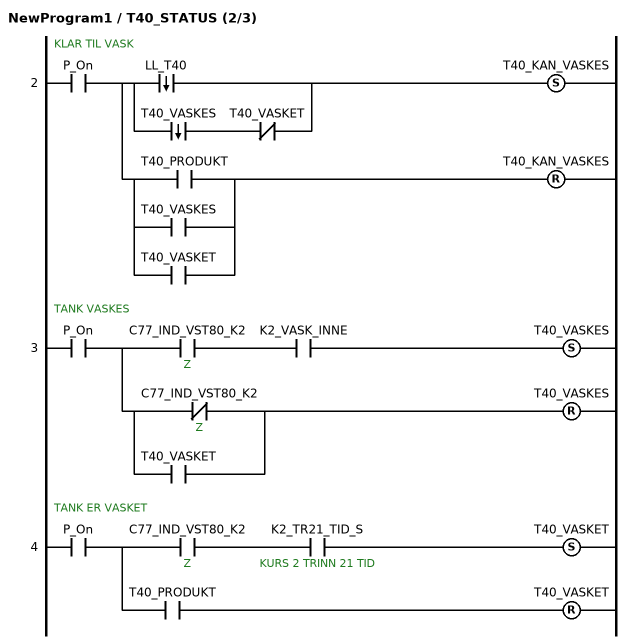
; [picture p1008: NewProgram1 / T40_STATUS, rungs 2-4]
; rung 2: KLAR TIL VASK
LD P_On
OUT TR0
%LD LL_T40
%LD T40_VASKES
ANDNOT T40_VASKET
ORLD
ANDLD
SET T40_KAN_VASKES
LD TR0
LD T40_PRODUKT
OR T40_VASKES
OR T40_VASKET
ANDLD
RSET T40_KAN_VASKES
; rung 3: TANK VASKES
LD P_On
OUT TR0
AND C77_IND_VST80_K2  ; Z
AND K2_VASK_INNE
SET T40_VASKES
LD TR0
LDNOT C77_IND_VST80_K2  ; Z
OR T40_VASKET
ANDLD
RSET T40_VASKES
; rung 4: TANK ER VASKET
LD P_On
OUT TR0
AND C77_IND_VST80_K2  ; Z
AND K2_TR21_TID_S  ; KURS 2 TRINN 21 TID
SET T40_VASKET
LD TR0
AND T40_PRODUKT
RSET T40_VASKET

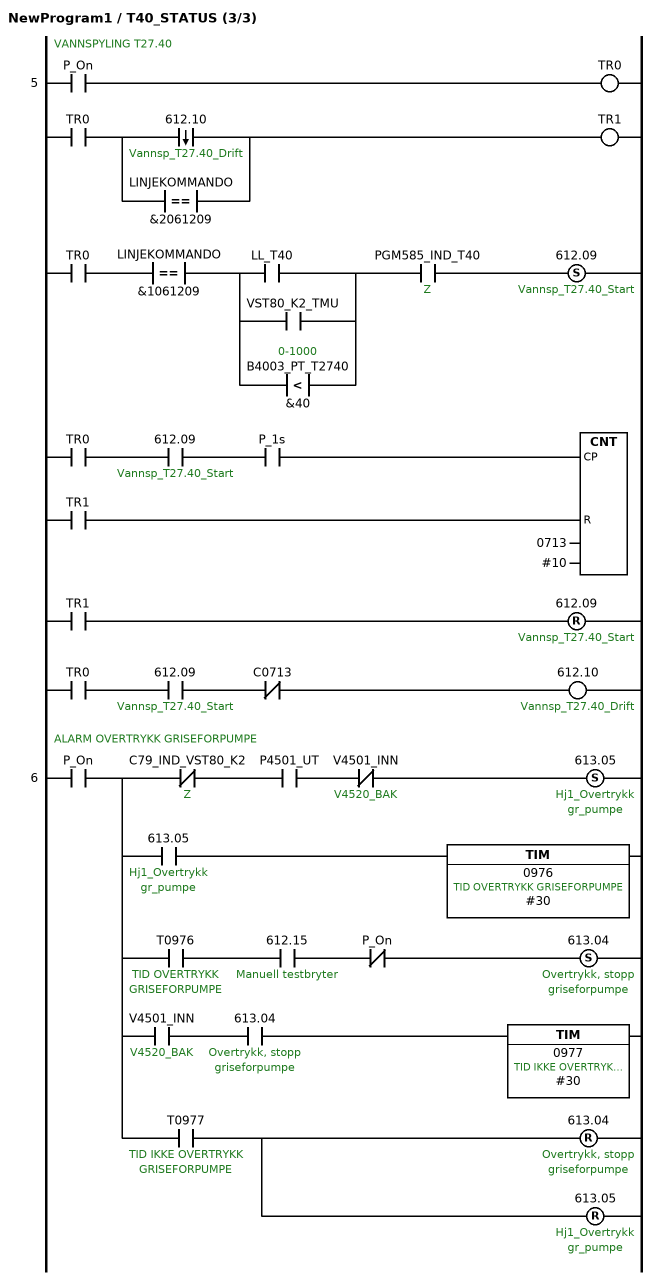
; rung 5: VANNSPYLING T27.40
LD P_On
OUT TR0
AND=L(301) LINJEKOMMANDO &1061209
LD LL_T40
OR VST80_K2_TMU
OR<(310) B4003_PT_T2740 &40  ; 0-1000
ANDLD
AND PGM585_IND_T40  ; Z
SET 612.09  ; Vannsp_T27.40_Start
LD TR0
AND 612.09  ; Vannsp_T27.40_Start
AND P_1s
LD TR0
%LD 612.10  ; Vannsp_T27.40_Drift
OR=L(301) LINJEKOMMANDO &2061209
ANDLD
OUT TR1
CNT 0713 #10
LD TR1
RSET 612.09  ; Vannsp_T27.40_Start
LD TR0
AND 612.09  ; Vannsp_T27.40_Start
ANDNOT C0713
OUT 612.10  ; Vannsp_T27.40_Drift
; rung 6: ALARM OVERTRYKK GRISEFORPUMPE
LD P_On
OUT TR0
ANDNOT C79_IND_VST80_K2  ; Z
AND P4501_UT
ANDNOT V4501_INN  ; V4520_BAK
SET 613.05  ; Hj1_Overtrykk gr_pumpe
LD TR0
AND 613.05  ; Hj1_Overtrykk gr_pumpe
TIM 0976 #30  ; TID OVERTRYKK GRISEFORPUMPE
LD TR0
AND T0976  ; TID OVERTRYKK GRISEFORPUMPE
AND 612.15  ; Manuell testbryter
ANDNOT P_On
SET 613.04  ; Overtrykk, stopp griseforpumpe
LD TR0
AND V4501_INN  ; V4520_BAK
AND 613.04  ; Overtrykk, stopp griseforpumpe
TIM 0977 #30  ; TID IKKE OVERTRYKK GRISEFORPUMPE
LD TR0
AND T0977  ; TID IKKE OVERTRYKK GRISEFORPUMPE
RSET 613.04  ; Overtrykk, stopp griseforpumpe
RSET 613.05  ; Hj1_Overtrykk gr_pumpe
; rung 7: Ingen_kommentar_funnet

### Section T40_VENTILER_RV_PUMPER

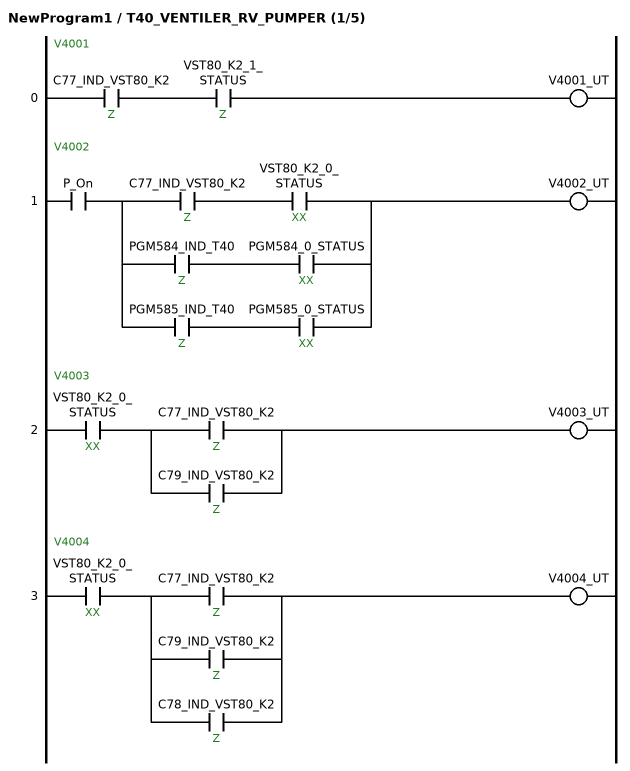
; rung 0: V4001
LD C77_IND_VST80_K2  ; Z
AND VST80_K2_1_STATUS  ; Z
OUT V4001_UT
; rung 1: V4002
LD P_On
LD C77_IND_VST80_K2  ; Z
AND VST80_K2_0_STATUS  ; XX
LD PGM584_IND_T40  ; Z
AND PGM584_0_STATUS  ; XX
ORLD
LD PGM585_IND_T40  ; Z
AND PGM585_0_STATUS  ; XX
ORLD
ANDLD
OUT V4002_UT
; rung 2: V4003
LD VST80_K2_0_STATUS  ; XX
LD C77_IND_VST80_K2  ; Z
OR C79_IND_VST80_K2  ; Z
ANDLD
OUT V4003_UT
; rung 3: V4004
LD VST80_K2_0_STATUS  ; XX
LD C77_IND_VST80_K2  ; Z
OR C79_IND_VST80_K2  ; Z
OR C78_IND_VST80_K2  ; Z
ANDLD
OUT V4004_UT

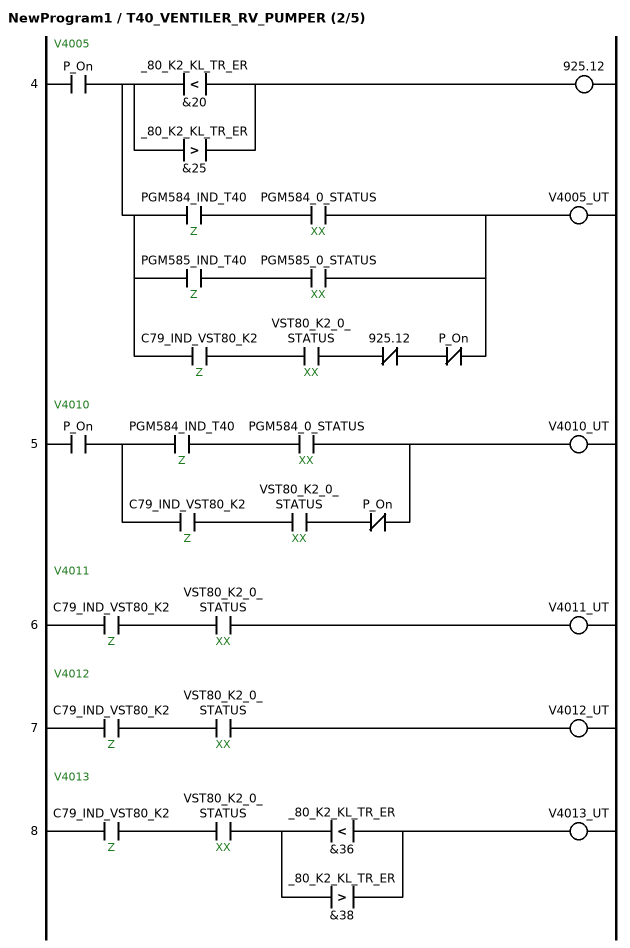
; rung 4: V4005
LD P_On
OUT TR0
LD<(310) _80_K2_KL_TR_ER &20
OR>(320) _80_K2_KL_TR_ER &25
ANDLD
OUT 925.12
LD TR0
LD PGM584_IND_T40  ; Z
AND PGM584_0_STATUS  ; XX
LD PGM585_IND_T40  ; Z
AND PGM585_0_STATUS  ; XX
ORLD
LD C79_IND_VST80_K2  ; Z
AND VST80_K2_0_STATUS  ; XX
ANDNOT 925.12
ANDNOT P_On
ORLD
ANDLD
OUT V4005_UT
; rung 5: V4010
LD P_On
LD PGM584_IND_T40  ; Z
AND PGM584_0_STATUS  ; XX
LD C79_IND_VST80_K2  ; Z
AND VST80_K2_0_STATUS  ; XX
ANDNOT P_On
ORLD
ANDLD
OUT V4010_UT
; rung 6: V4011
LD C79_IND_VST80_K2  ; Z
AND VST80_K2_0_STATUS  ; XX
OUT V4011_UT
; rung 7: V4012
LD C79_IND_VST80_K2  ; Z
AND VST80_K2_0_STATUS  ; XX
OUT V4012_UT
; rung 8: V4013
LD C79_IND_VST80_K2  ; Z
AND VST80_K2_0_STATUS  ; XX
LD<(310) _80_K2_KL_TR_ER &36
OR>(320) _80_K2_KL_TR_ER &38
ANDLD
OUT V4013_UT

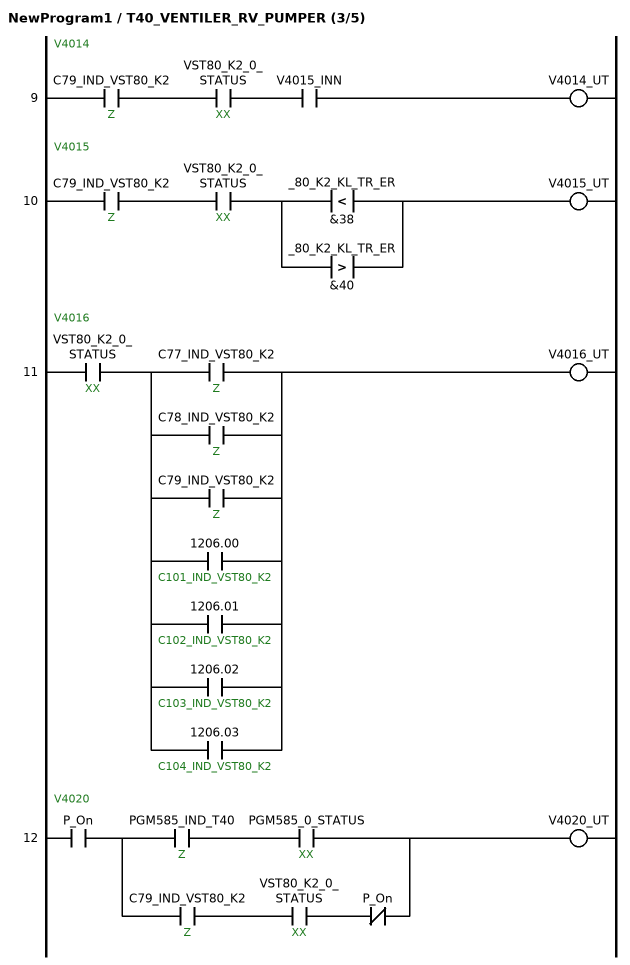
; rung 9: V4014
LD C79_IND_VST80_K2  ; Z
AND VST80_K2_0_STATUS  ; XX
AND V4015_INN
OUT V4014_UT
; rung 10: V4015
LD C79_IND_VST80_K2  ; Z
AND VST80_K2_0_STATUS  ; XX
LD<(310) _80_K2_KL_TR_ER &38
OR>(320) _80_K2_KL_TR_ER &40
ANDLD
OUT V4015_UT
; rung 11: V4016
LD VST80_K2_0_STATUS  ; XX
LD C77_IND_VST80_K2  ; Z
OR C78_IND_VST80_K2  ; Z
OR C79_IND_VST80_K2  ; Z
OR 1206.00  ; C101_IND_VST80_K2
OR 1206.01  ; C102_IND_VST80_K2
OR 1206.02  ; C103_IND_VST80_K2
OR 1206.03  ; C104_IND_VST80_K2
ANDLD
OUT V4016_UT
; rung 12: V4020
LD P_On
LD PGM585_IND_T40  ; Z
AND PGM585_0_STATUS  ; XX
LD C79_IND_VST80_K2  ; Z
AND VST80_K2_0_STATUS  ; XX
ANDNOT P_On
ORLD
ANDLD
OUT V4020_UT

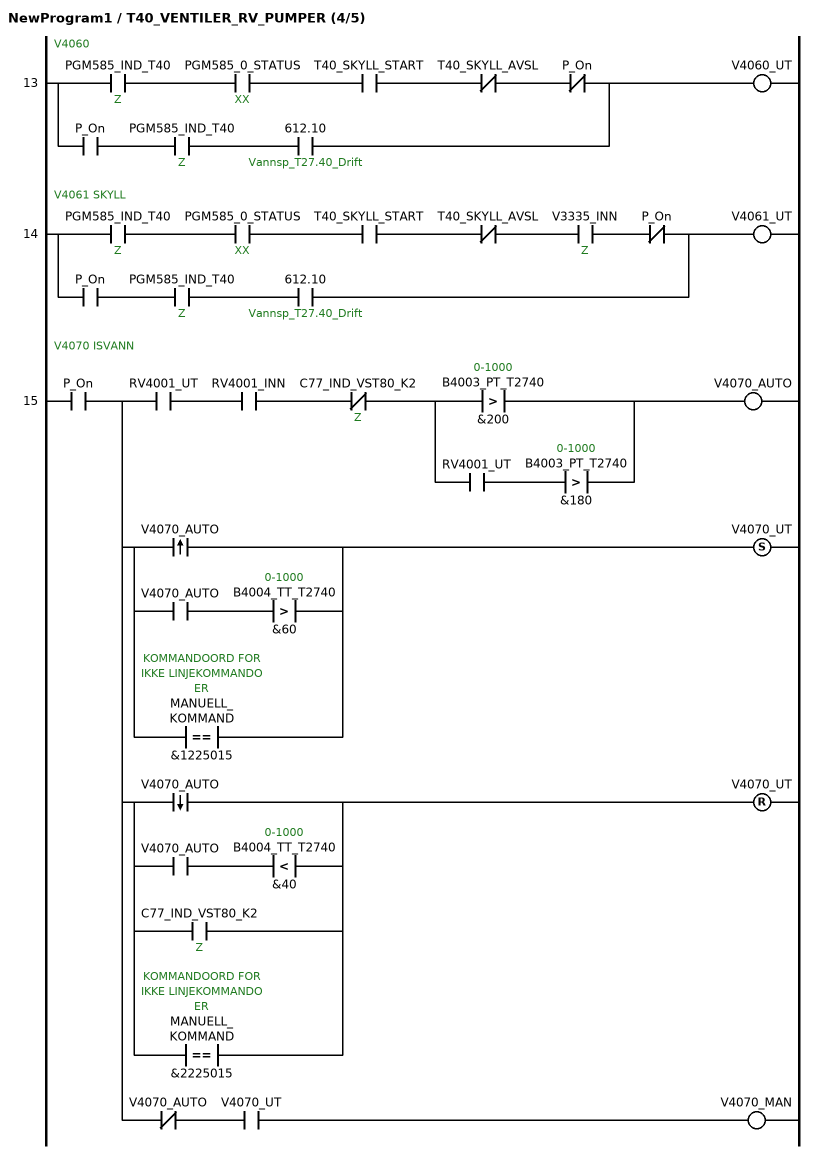
; rung 13: V4060
LD PGM585_IND_T40  ; Z
AND PGM585_0_STATUS  ; XX
AND T40_SKYLL_START
ANDNOT T40_SKYLL_AVSL
ANDNOT P_On
LD P_On
AND PGM585_IND_T40  ; Z
AND 612.10  ; Vannsp_T27.40_Drift
ORLD
OUT V4060_UT
; rung 14: V4061 SKYLL
LD PGM585_IND_T40  ; Z
AND PGM585_0_STATUS  ; XX
AND T40_SKYLL_START
ANDNOT T40_SKYLL_AVSL
AND V3335_INN  ; Z
ANDNOT P_On
LD P_On
AND PGM585_IND_T40  ; Z
AND 612.10  ; Vannsp_T27.40_Drift
ORLD
OUT V4061_UT
; rung 15: V4070 ISVANN
LD P_On
OUT TR0
AND RV4001_UT
AND RV4001_INN
ANDNOT C77_IND_VST80_K2  ; Z
LD>(320) B4003_PT_T2740 &200  ; 0-1000
LD RV4001_UT
AND>(320) B4003_PT_T2740 &180  ; 0-1000
ORLD
ANDLD
OUT V4070_AUTO
LD TR0
@LD V4070_AUTO
LD V4070_AUTO
AND>(320) B4004_TT_T2740 &60  ; 0-1000
ORLD
OR=L(301) MANUELL_KOMMAND &1225015  ; KOMMANDOORD FOR IKKE LINJEKOMMANDOER
ANDLD
SET V4070_UT
LD TR0
%LD V4070_AUTO
LD V4070_AUTO
AND<(310) B4004_TT_T2740 &40  ; 0-1000
ORLD
OR C77_IND_VST80_K2  ; Z
OR=L(301) MANUELL_KOMMAND &2225015  ; KOMMANDOORD FOR IKKE LINJEKOMMANDOER
ANDLD
RSET V4070_UT
LD TR0
ANDNOT V4070_AUTO
AND V4070_UT
OUT V4070_MAN

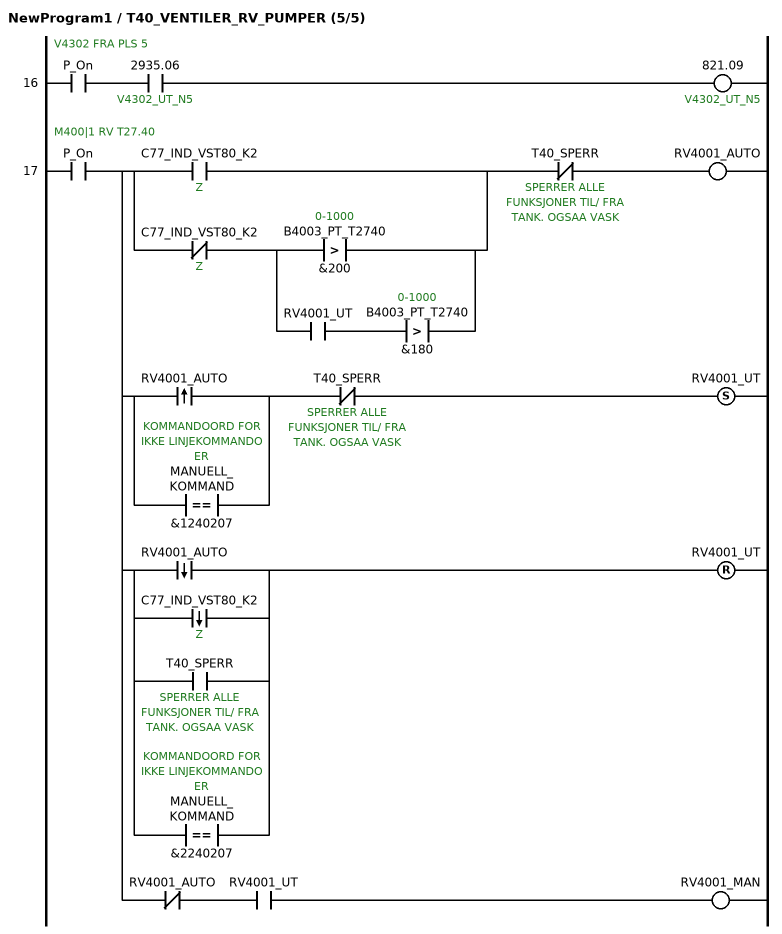
; rung 16: V4302 FRA PLS 5
LD P_On
AND 2935.06  ; V4302_UT_N5
OUT 821.09  ; V4302_UT_N5
; rung 17: M400|1 RV T27.40
LD P_On
OUT TR0
LD C77_IND_VST80_K2  ; Z
LDNOT C77_IND_VST80_K2  ; Z
LD>(320) B4003_PT_T2740 &200  ; 0-1000
LD RV4001_UT
AND>(320) B4003_PT_T2740 &180  ; 0-1000
ORLD
ANDLD
ORLD
ANDLD
ANDNOT T40_SPERR  ; SPERRER ALLE FUNKSJONER TIL/ FRA TANK. OGSAA VASK
OUT RV4001_AUTO
LD TR0
@LD RV4001_AUTO
OR=L(301) MANUELL_KOMMAND &1240207  ; KOMMANDOORD FOR IKKE LINJEKOMMANDOER
ANDLD
ANDNOT T40_SPERR  ; SPERRER ALLE FUNKSJONER TIL/ FRA TANK. OGSAA VASK
SET RV4001_UT
LD TR0
%LD RV4001_AUTO
%OR C77_IND_VST80_K2  ; Z
OR T40_SPERR  ; SPERRER ALLE FUNKSJONER TIL/ FRA TANK. OGSAA VASK
OR=L(301) MANUELL_KOMMAND &2240207  ; KOMMANDOORD FOR IKKE LINJEKOMMANDOER
ANDLD
RSET RV4001_UT
LD TR0
ANDNOT RV4001_AUTO
AND RV4001_UT
OUT RV4001_MAN
; rung 18: Ingen_kommentar_funnet

### Section T41_TEMP_NIVÅ

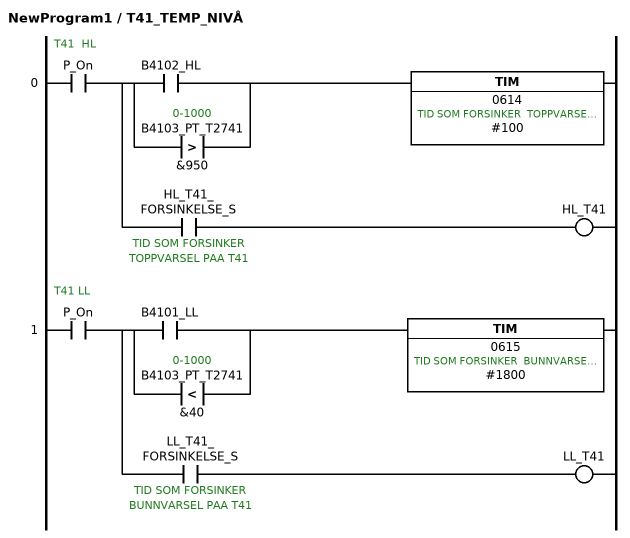
; rung 0: T41  HL
LD P_On
OUT TR0
LD B4102_HL
OR>(320) B4103_PT_T2741 &950  ; 0-1000
ANDLD
TIM 0614 #100  ; TID SOM FORSINKER  TOPPVARSEL PAA T41
LD TR0
AND HL_T41_FORSINKELSE_S  ; TID SOM FORSINKER  TOPPVARSEL PAA T41
OUT HL_T41
; rung 1: T41 LL
LD P_On
OUT TR0
LD B4101_LL
OR<(310) B4103_PT_T2741 &40  ; 0-1000
ANDLD
TIM 0615 #1800  ; TID SOM FORSINKER  BUNNVARSEL PAA T41
LD TR0
AND LL_T41_FORSINKELSE_S  ; TID SOM FORSINKER  BUNNVARSEL PAA T41
OUT LL_T41
; rung 2: Ingen_kommentar_funnet

### Section T41_STATUS

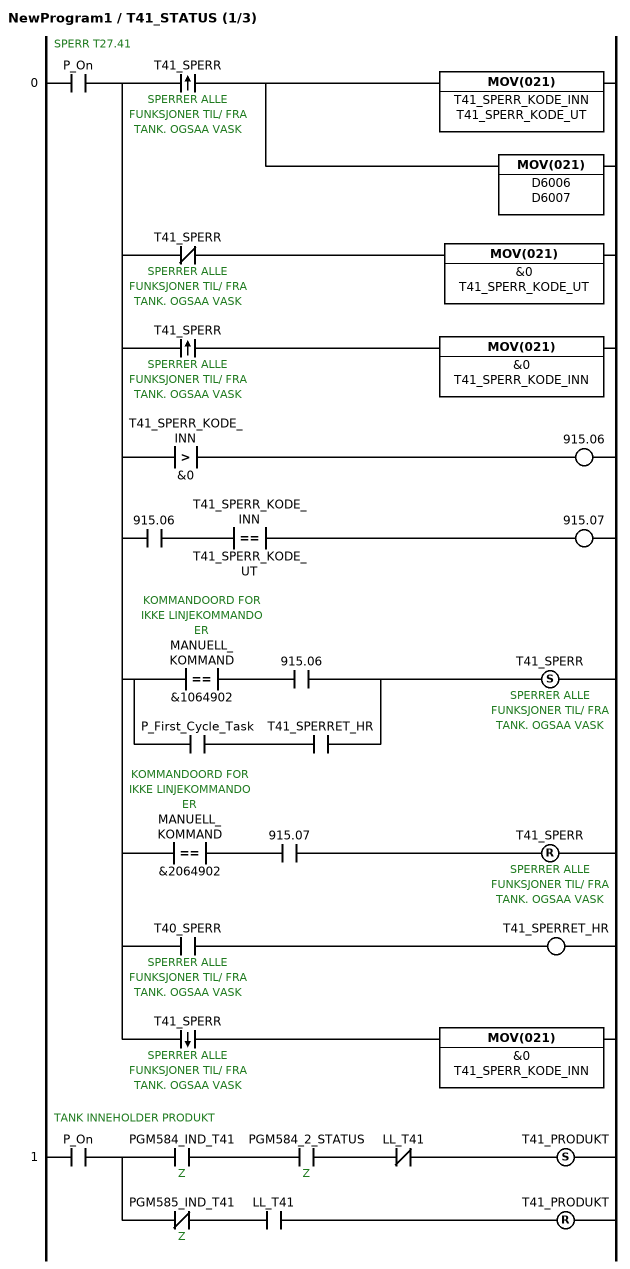
; rung 0: SPERR T27.41
LD P_On
OUT TR0
@AND T41_SPERR  ; SPERRER ALLE FUNKSJONER TIL/ FRA TANK. OGSAA VASK
MOV(021) T41_SPERR_KODE_INN T41_SPERR_KODE_UT
MOV(021) D6006 D6007
LD TR0
ANDNOT T41_SPERR  ; SPERRER ALLE FUNKSJONER TIL/ FRA TANK. OGSAA VASK
MOV(021) &0 T41_SPERR_KODE_UT
LD TR0
@AND T41_SPERR  ; SPERRER ALLE FUNKSJONER TIL/ FRA TANK. OGSAA VASK
MOV(021) &0 T41_SPERR_KODE_INN
LD TR0
AND>(320) T41_SPERR_KODE_INN &0
OUT 915.06
LD TR0
AND 915.06
AND=(300) T41_SPERR_KODE_INN T41_SPERR_KODE_UT
OUT 915.07
LD TR0
LD=L(301) MANUELL_KOMMAND &1064902  ; KOMMANDOORD FOR IKKE LINJEKOMMANDOER
AND 915.06
LD P_First_Cycle_Task
AND T41_SPERRET_HR
ORLD
ANDLD
SET T41_SPERR  ; SPERRER ALLE FUNKSJONER TIL/ FRA TANK. OGSAA VASK
LD TR0
AND=L(301) MANUELL_KOMMAND &2064902  ; KOMMANDOORD FOR IKKE LINJEKOMMANDOER
AND 915.07
RSET T41_SPERR  ; SPERRER ALLE FUNKSJONER TIL/ FRA TANK. OGSAA VASK
LD TR0
AND T40_SPERR  ; SPERRER ALLE FUNKSJONER TIL/ FRA TANK. OGSAA VASK
OUT T41_SPERRET_HR
LD TR0
%AND T41_SPERR  ; SPERRER ALLE FUNKSJONER TIL/ FRA TANK. OGSAA VASK
MOV(021) &0 T41_SPERR_KODE_INN
; rung 1: TANK INNEHOLDER PRODUKT
LD P_On
OUT TR0
AND PGM584_IND_T41  ; Z
AND PGM584_2_STATUS  ; Z
ANDNOT LL_T41
SET T41_PRODUKT
LD TR0
ANDNOT PGM585_IND_T41  ; Z
AND LL_T41
RSET T41_PRODUKT

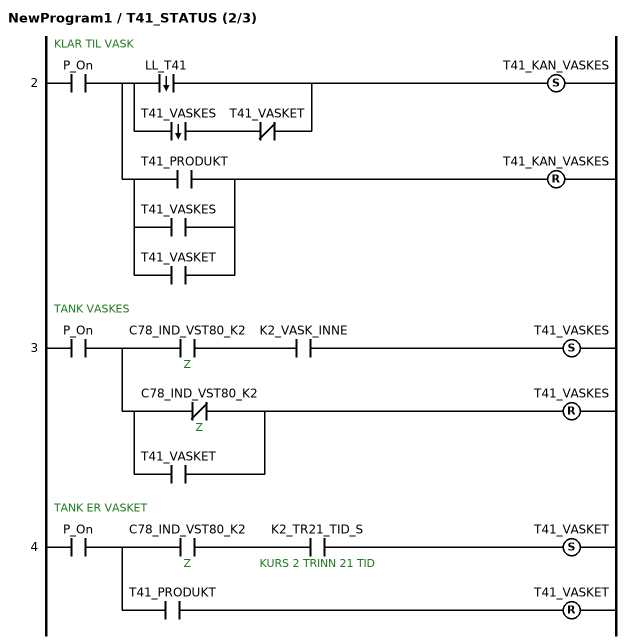
; rung 2: KLAR TIL VASK
LD P_On
OUT TR0
%LD LL_T41
%LD T41_VASKES
ANDNOT T41_VASKET
ORLD
ANDLD
SET T41_KAN_VASKES
LD TR0
LD T41_PRODUKT
OR T41_VASKES
OR T41_VASKET
ANDLD
RSET T41_KAN_VASKES
; rung 3: TANK VASKES
LD P_On
OUT TR0
AND C78_IND_VST80_K2  ; Z
AND K2_VASK_INNE
SET T41_VASKES
LD TR0
LDNOT C78_IND_VST80_K2  ; Z
OR T41_VASKET
ANDLD
RSET T41_VASKES
; rung 4: TANK ER VASKET
LD P_On
OUT TR0
AND C78_IND_VST80_K2  ; Z
AND K2_TR21_TID_S  ; KURS 2 TRINN 21 TID
SET T41_VASKET
LD TR0
AND T41_PRODUKT
RSET T41_VASKET

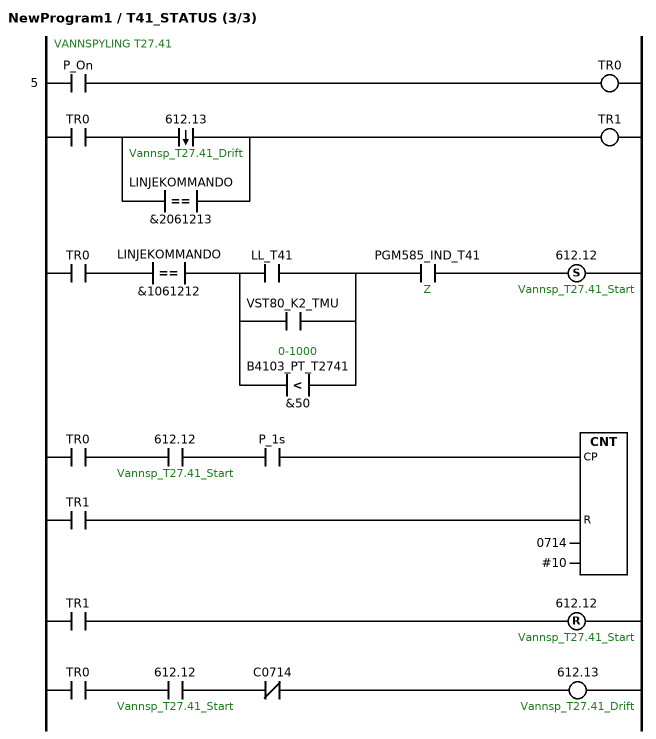
; rung 5: VANNSPYLING T27.41
LD P_On
OUT TR0
AND=L(301) LINJEKOMMANDO &1061212
LD LL_T41
OR VST80_K2_TMU
OR<(310) B4103_PT_T2741 &50  ; 0-1000
ANDLD
AND PGM585_IND_T41  ; Z
SET 612.12  ; Vannsp_T27.41_Start
LD TR0
AND 612.12  ; Vannsp_T27.41_Start
AND P_1s
LD TR0
%LD 612.13  ; Vannsp_T27.41_Drift
OR=L(301) LINJEKOMMANDO &2061213
ANDLD
OUT TR1
CNT 0714 #10
LD TR1
RSET 612.12  ; Vannsp_T27.41_Start
LD TR0
AND 612.12  ; Vannsp_T27.41_Start
ANDNOT C0714
OUT 612.13  ; Vannsp_T27.41_Drift
; rung 6: Ingen_kommentar_funnet

### Section T41_VENTILER_RV_PUMPER

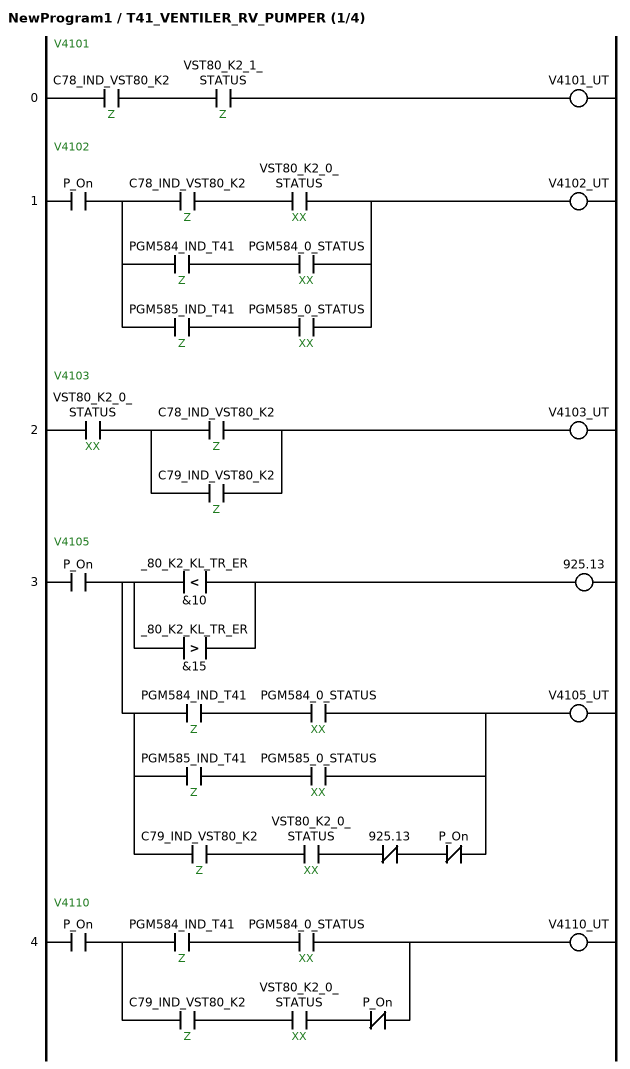
; rung 0: V4101
LD C78_IND_VST80_K2  ; Z
AND VST80_K2_1_STATUS  ; Z
OUT V4101_UT
; rung 1: V4102
LD P_On
LD C78_IND_VST80_K2  ; Z
AND VST80_K2_0_STATUS  ; XX
LD PGM584_IND_T41  ; Z
AND PGM584_0_STATUS  ; XX
ORLD
LD PGM585_IND_T41  ; Z
AND PGM585_0_STATUS  ; XX
ORLD
ANDLD
OUT V4102_UT
; rung 2: V4103
LD VST80_K2_0_STATUS  ; XX
LD C78_IND_VST80_K2  ; Z
OR C79_IND_VST80_K2  ; Z
ANDLD
OUT V4103_UT
; rung 3: V4105
LD P_On
OUT TR0
LD<(310) _80_K2_KL_TR_ER &10
OR>(320) _80_K2_KL_TR_ER &15
ANDLD
OUT 925.13
LD TR0
LD PGM584_IND_T41  ; Z
AND PGM584_0_STATUS  ; XX
LD PGM585_IND_T41  ; Z
AND PGM585_0_STATUS  ; XX
ORLD
LD C79_IND_VST80_K2  ; Z
AND VST80_K2_0_STATUS  ; XX
ANDNOT 925.13
ANDNOT P_On
ORLD
ANDLD
OUT V4105_UT
; rung 4: V4110
LD P_On
LD PGM584_IND_T41  ; Z
AND PGM584_0_STATUS  ; XX
LD C79_IND_VST80_K2  ; Z
AND VST80_K2_0_STATUS  ; XX
ANDNOT P_On
ORLD
ANDLD
OUT V4110_UT

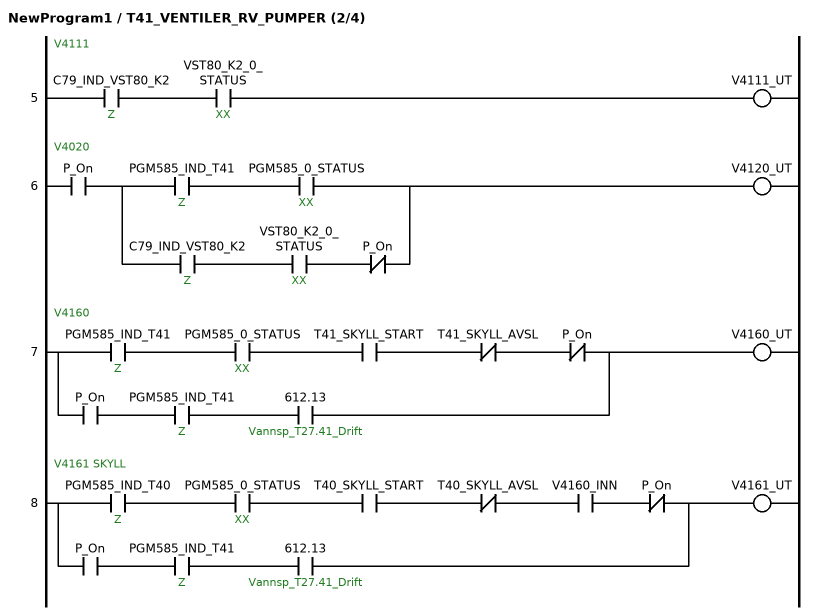
; rung 5: V4111
LD C79_IND_VST80_K2  ; Z
AND VST80_K2_0_STATUS  ; XX
OUT V4111_UT
; rung 6: V4020
LD P_On
LD PGM585_IND_T41  ; Z
AND PGM585_0_STATUS  ; XX
LD C79_IND_VST80_K2  ; Z
AND VST80_K2_0_STATUS  ; XX
ANDNOT P_On
ORLD
ANDLD
OUT V4120_UT
; rung 7: V4160
LD PGM585_IND_T41  ; Z
AND PGM585_0_STATUS  ; XX
AND T41_SKYLL_START
ANDNOT T41_SKYLL_AVSL
ANDNOT P_On
LD P_On
AND PGM585_IND_T41  ; Z
AND 612.13  ; Vannsp_T27.41_Drift
ORLD
OUT V4160_UT
; rung 8: V4161 SKYLL
LD PGM585_IND_T40  ; Z
AND PGM585_0_STATUS  ; XX
AND T40_SKYLL_START
ANDNOT T40_SKYLL_AVSL
AND V4160_INN
ANDNOT P_On
LD P_On
AND PGM585_IND_T41  ; Z
AND 612.13  ; Vannsp_T27.41_Drift
ORLD
OUT V4161_UT

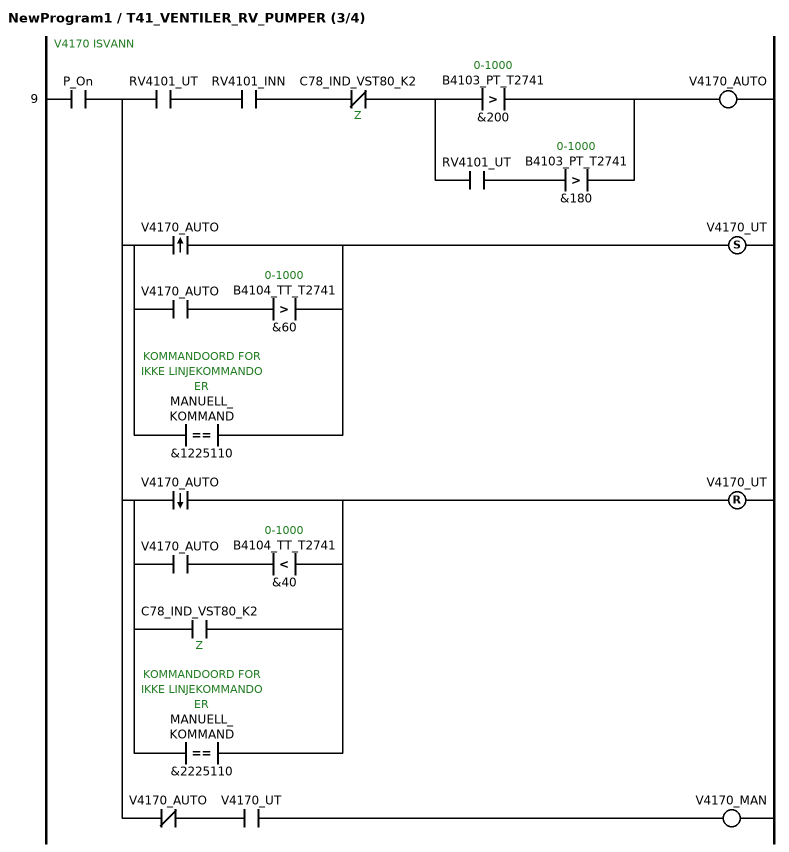
; rung 9: V4170 ISVANN
LD P_On
OUT TR0
AND RV4101_UT
AND RV4101_INN
ANDNOT C78_IND_VST80_K2  ; Z
LD>(320) B4103_PT_T2741 &200  ; 0-1000
LD RV4101_UT
AND>(320) B4103_PT_T2741 &180  ; 0-1000
ORLD
ANDLD
OUT V4170_AUTO
LD TR0
@LD V4170_AUTO
LD V4170_AUTO
AND>(320) B4104_TT_T2741 &60  ; 0-1000
ORLD
OR=L(301) MANUELL_KOMMAND &1225110  ; KOMMANDOORD FOR IKKE LINJEKOMMANDOER
ANDLD
SET V4170_UT
LD TR0
%LD V4170_AUTO
LD V4170_AUTO
AND<(310) B4104_TT_T2741 &40  ; 0-1000
ORLD
OR C78_IND_VST80_K2  ; Z
OR=L(301) MANUELL_KOMMAND &2225110  ; KOMMANDOORD FOR IKKE LINJEKOMMANDOER
ANDLD
RSET V4170_UT
LD TR0
ANDNOT V4170_AUTO
AND V4170_UT
OUT V4170_MAN

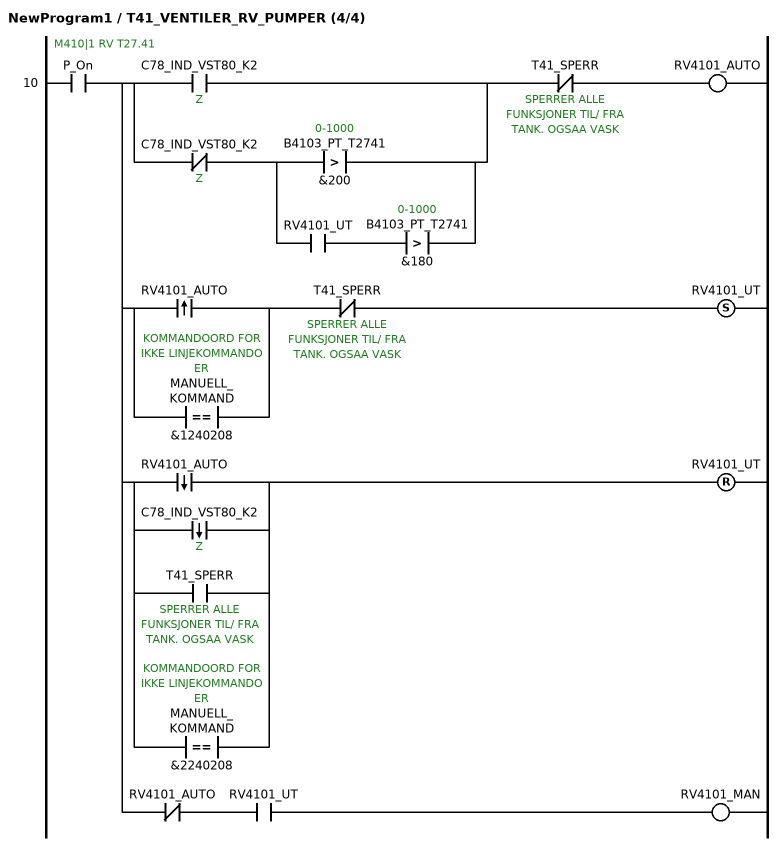
; rung 10: M410|1 RV T27.41
LD P_On
OUT TR0
LD C78_IND_VST80_K2  ; Z
LDNOT C78_IND_VST80_K2  ; Z
LD>(320) B4103_PT_T2741 &200  ; 0-1000
LD RV4101_UT
AND>(320) B4103_PT_T2741 &180  ; 0-1000
ORLD
ANDLD
ORLD
ANDLD
ANDNOT T41_SPERR  ; SPERRER ALLE FUNKSJONER TIL/ FRA TANK. OGSAA VASK
OUT RV4101_AUTO
LD TR0
@LD RV4101_AUTO
OR=L(301) MANUELL_KOMMAND &1240208  ; KOMMANDOORD FOR IKKE LINJEKOMMANDOER
ANDLD
ANDNOT T41_SPERR  ; SPERRER ALLE FUNKSJONER TIL/ FRA TANK. OGSAA VASK
SET RV4101_UT
LD TR0
%LD RV4101_AUTO
%OR C78_IND_VST80_K2  ; Z
OR T41_SPERR  ; SPERRER ALLE FUNKSJONER TIL/ FRA TANK. OGSAA VASK
OR=L(301) MANUELL_KOMMAND &2240208  ; KOMMANDOORD FOR IKKE LINJEKOMMANDOER
ANDLD
RSET RV4101_UT
LD TR0
ANDNOT RV4101_AUTO
AND RV4101_UT
OUT RV4101_MAN
; rung 11: Ingen_kommentar_funnet

### Section T43_GR44_T45_VENTILER_PUMPER

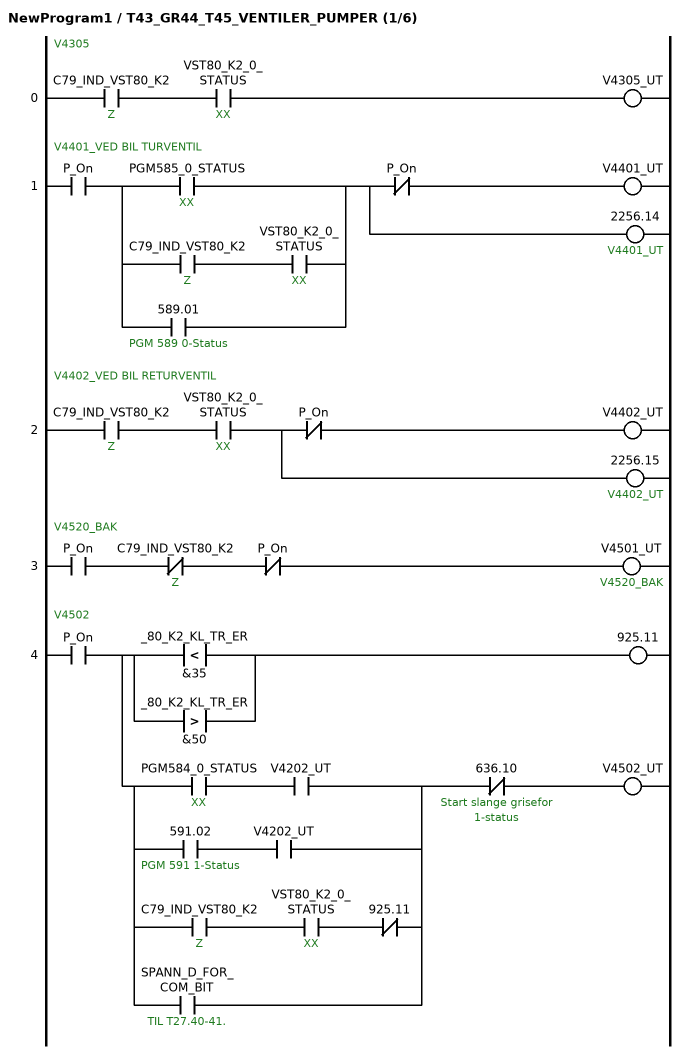
; rung 0: V4305
LD C79_IND_VST80_K2  ; Z
AND VST80_K2_0_STATUS  ; XX
OUT V4305_UT
; rung 1: V4401_VED BIL TURVENTIL
LD P_On
LD PGM585_0_STATUS  ; XX
LD C79_IND_VST80_K2  ; Z
AND VST80_K2_0_STATUS  ; XX
ORLD
OR 589.01  ; PGM 589 0-Status
ANDLD
OUT TR0
ANDNOT P_On
OUT V4401_UT
LD TR0
OUT 2256.14  ; V4401_UT
; rung 2: V4402_VED BIL RETURVENTIL
LD C79_IND_VST80_K2  ; Z
AND VST80_K2_0_STATUS  ; XX
OUT TR0
ANDNOT P_On
OUT V4402_UT
LD TR0
OUT 2256.15  ; V4402_UT
; rung 3: V4520_BAK
LD P_On
ANDNOT C79_IND_VST80_K2  ; Z
ANDNOT P_On
OUT V4501_UT  ; V4520_BAK
; rung 4: V4502
LD P_On
OUT TR0
LD<(310) _80_K2_KL_TR_ER &35
OR>(320) _80_K2_KL_TR_ER &50
ANDLD
OUT 925.11
LD TR0
LD PGM584_0_STATUS  ; XX
AND V4202_UT
LD 591.02  ; PGM 591 1-Status
AND V4202_UT
ORLD
LD C79_IND_VST80_K2  ; Z
AND VST80_K2_0_STATUS  ; XX
ANDNOT 925.11
ORLD
OR SPANN_D_FOR_COM_BIT  ; TIL T27.40-41.
ANDLD
ANDNOT 636.10  ; Start slange grisefor 1-status
OUT V4502_UT

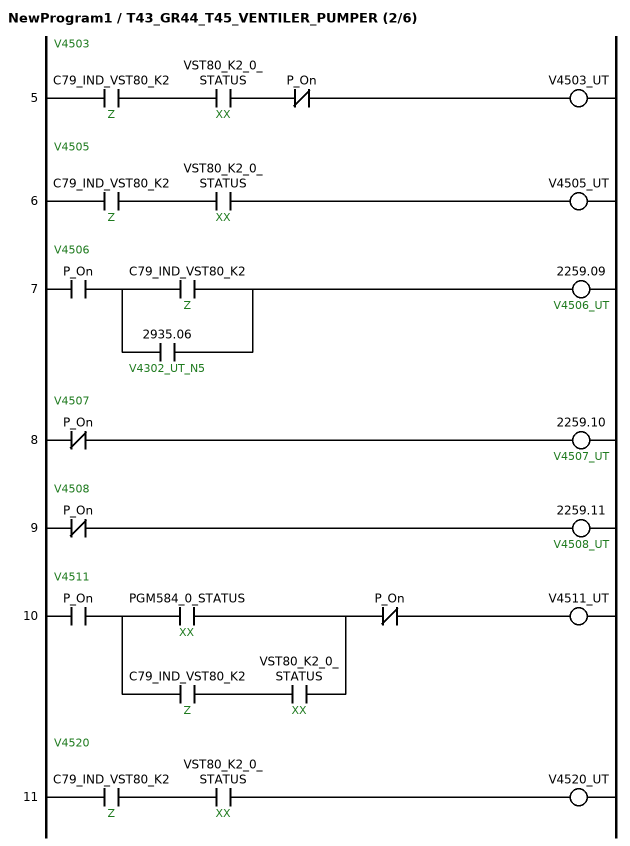
; rung 5: V4503
LD C79_IND_VST80_K2  ; Z
AND VST80_K2_0_STATUS  ; XX
ANDNOT P_On
OUT V4503_UT
; rung 6: V4505
LD C79_IND_VST80_K2  ; Z
AND VST80_K2_0_STATUS  ; XX
OUT V4505_UT
; rung 7: V4506
LD P_On
LD C79_IND_VST80_K2  ; Z
OR 2935.06  ; V4302_UT_N5
ANDLD
OUT 2259.09  ; V4506_UT
; rung 8: V4507
LDNOT P_On
OUT 2259.10  ; V4507_UT
; rung 9: V4508
LDNOT P_On
OUT 2259.11  ; V4508_UT
; rung 10: V4511
LD P_On
LD PGM584_0_STATUS  ; XX
LD C79_IND_VST80_K2  ; Z
AND VST80_K2_0_STATUS  ; XX
ORLD
ANDLD
ANDNOT P_On
OUT V4511_UT
; rung 11: V4520
LD C79_IND_VST80_K2  ; Z
AND VST80_K2_0_STATUS  ; XX
OUT V4520_UT

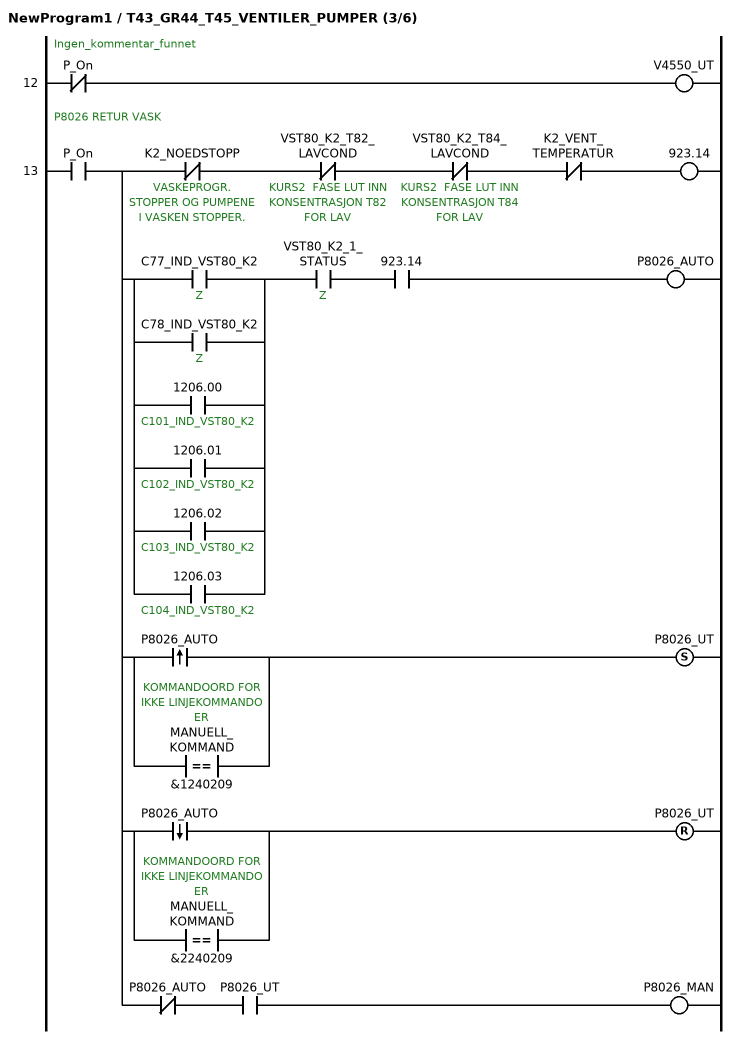
; rung 12: Ingen_kommentar_funnet
LDNOT P_On
OUT V4550_UT
; rung 13: P8026 RETUR VASK
LD P_On
OUT TR0
ANDNOT K2_NOEDSTOPP  ; VASKEPROGR. STOPPER OG PUMPENE I VASKEN STOPPER.
ANDNOT VST80_K2_T82_LAVCOND  ; KURS2  FASE LUT INN KONSENTRASJON T82 FOR LAV
ANDNOT VST80_K2_T84_LAVCOND  ; KURS2  FASE LUT INN KONSENTRASJON T84 FOR LAV
ANDNOT K2_VENT_TEMPERATUR
OUT 923.14
LD TR0
LD C77_IND_VST80_K2  ; Z
OR C78_IND_VST80_K2  ; Z
OR 1206.00  ; C101_IND_VST80_K2
OR 1206.01  ; C102_IND_VST80_K2
OR 1206.02  ; C103_IND_VST80_K2
OR 1206.03  ; C104_IND_VST80_K2
ANDLD
AND VST80_K2_1_STATUS  ; Z
AND 923.14
OUT P8026_AUTO
LD TR0
@LD P8026_AUTO
OR=L(301) MANUELL_KOMMAND &1240209  ; KOMMANDOORD FOR IKKE LINJEKOMMANDOER
ANDLD
SET P8026_UT
LD TR0
%LD P8026_AUTO
OR=L(301) MANUELL_KOMMAND &2240209  ; KOMMANDOORD FOR IKKE LINJEKOMMANDOER
ANDLD
RSET P8026_UT
LD TR0
ANDNOT P8026_AUTO
AND P8026_UT
OUT P8026_MAN

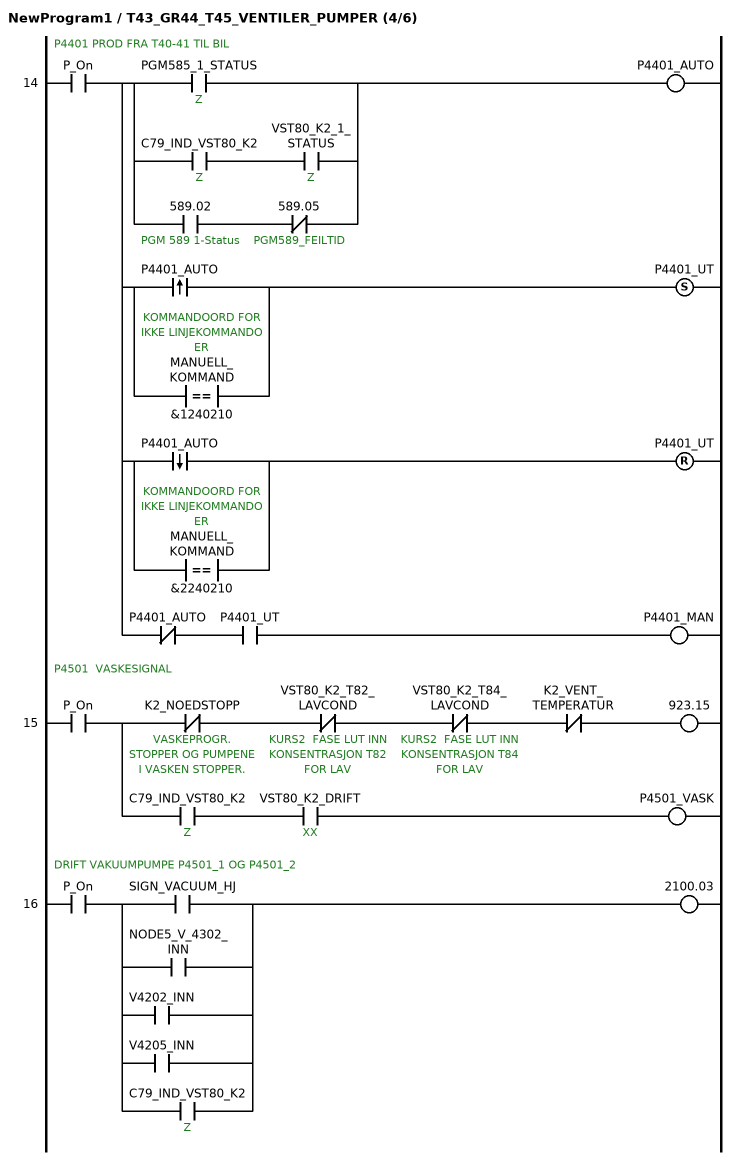
; rung 14: P4401 PROD FRA T40-41 TIL BIL
LD P_On
OUT TR0
LD PGM585_1_STATUS  ; Z
LD C79_IND_VST80_K2  ; Z
AND VST80_K2_1_STATUS  ; Z
ORLD
LD 589.02  ; PGM 589 1-Status
ANDNOT 589.05  ; PGM589_FEILTID
ORLD
ANDLD
OUT P4401_AUTO
LD TR0
@LD P4401_AUTO
OR=L(301) MANUELL_KOMMAND &1240210  ; KOMMANDOORD FOR IKKE LINJEKOMMANDOER
ANDLD
SET P4401_UT
LD TR0
%LD P4401_AUTO
OR=L(301) MANUELL_KOMMAND &2240210  ; KOMMANDOORD FOR IKKE LINJEKOMMANDOER
ANDLD
RSET P4401_UT
LD TR0
ANDNOT P4401_AUTO
AND P4401_UT
OUT P4401_MAN
; rung 15: P4501  VASKESIGNAL
LD P_On
OUT TR0
ANDNOT K2_NOEDSTOPP  ; VASKEPROGR. STOPPER OG PUMPENE I VASKEN STOPPER.
ANDNOT VST80_K2_T82_LAVCOND  ; KURS2  FASE LUT INN KONSENTRASJON T82 FOR LAV
ANDNOT VST80_K2_T84_LAVCOND  ; KURS2  FASE LUT INN KONSENTRASJON T84 FOR LAV
ANDNOT K2_VENT_TEMPERATUR
OUT 923.15
LD TR0
AND C79_IND_VST80_K2  ; Z
AND VST80_K2_DRIFT  ; XX
OUT P4501_VASK
; rung 16: DRIFT VAKUUMPUMPE P4501_1 OG P4501_2
LD P_On
LD SIGN_VACUUM_HJ
OR NODE5_V_4302_INN
OR V4202_INN
OR V4205_INN
OR C79_IND_VST80_K2  ; Z
ANDLD
OUT 2100.03

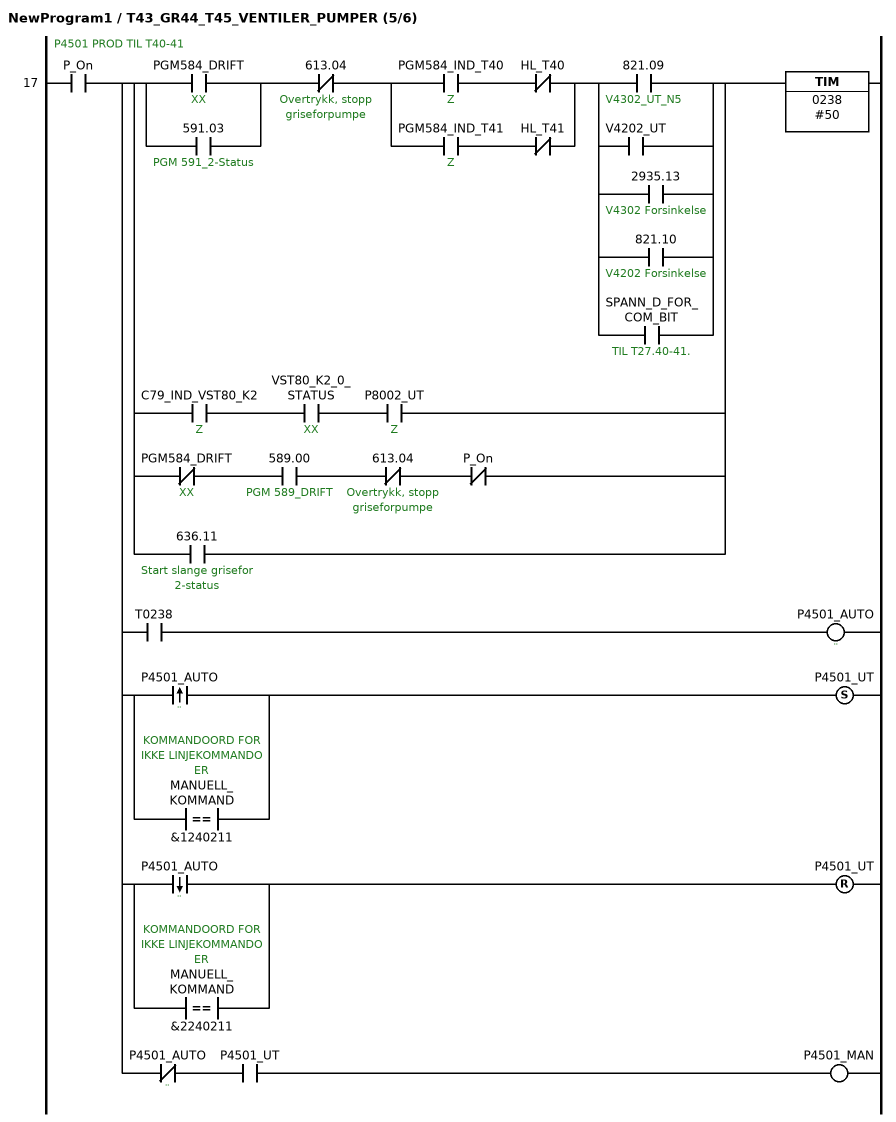
; rung 17: P4501 PROD TIL T40-41
LD P_On
OUT TR0
LD PGM584_DRIFT  ; XX
OR 591.03  ; PGM 591_2-Status
ANDNOT 613.04  ; Overtrykk, stopp griseforpumpe
LD PGM584_IND_T40  ; Z
ANDNOT HL_T40
LD PGM584_IND_T41  ; Z
ANDNOT HL_T41
ORLD
ANDLD
LD 821.09  ; V4302_UT_N5
OR V4202_UT
OR 2935.13  ; V4302 Forsinkelse
OR 821.10  ; V4202 Forsinkelse
OR SPANN_D_FOR_COM_BIT  ; TIL T27.40-41.
ANDLD
LD C79_IND_VST80_K2  ; Z
AND VST80_K2_0_STATUS  ; XX
AND P8002_UT  ; Z
ORLD
LDNOT PGM584_DRIFT  ; XX
AND 589.00  ; PGM 589_DRIFT
ANDNOT 613.04  ; Overtrykk, stopp griseforpumpe
ANDNOT P_On
ORLD
OR 636.11  ; Start slange grisefor 2-status
ANDLD
TIM 0238 #50
LD TR0
AND T0238
OUT P4501_AUTO  ; ¨
LD TR0
@LD P4501_AUTO  ; ¨
OR=L(301) MANUELL_KOMMAND &1240211  ; KOMMANDOORD FOR IKKE LINJEKOMMANDOER
ANDLD
SET P4501_UT
LD TR0
%LD P4501_AUTO  ; ¨
OR=L(301) MANUELL_KOMMAND &2240211  ; KOMMANDOORD FOR IKKE LINJEKOMMANDOER
ANDLD
RSET P4501_UT
LD TR0
ANDNOT P4501_AUTO  ; ¨
AND P4501_UT
OUT P4501_MAN

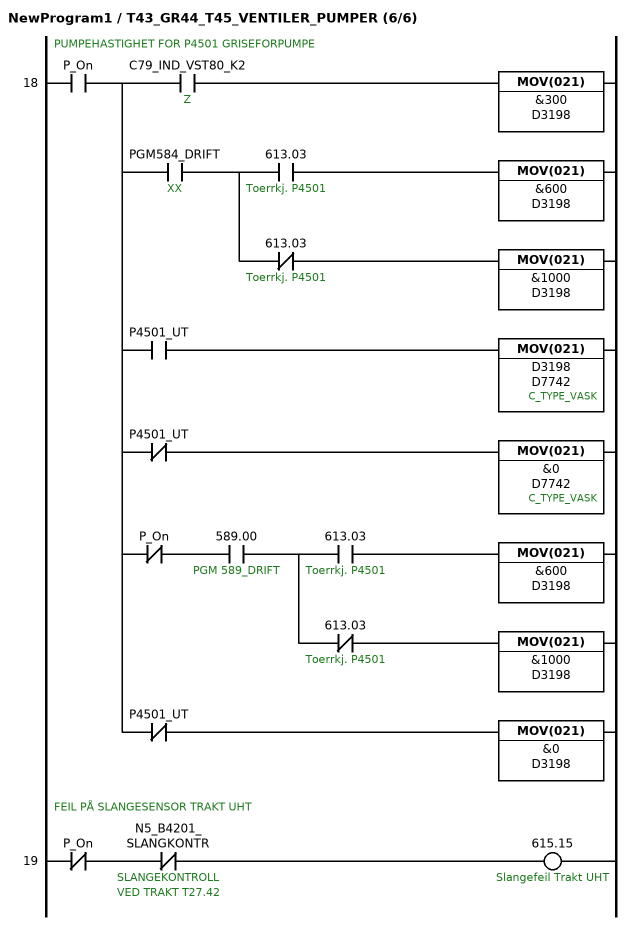
; rung 18: PUMPEHASTIGHET FOR P4501 GRISEFORPUMPE
LD P_On
OUT TR0
AND C79_IND_VST80_K2  ; Z
MOV(021) &300 D3198
LD TR0
AND PGM584_DRIFT  ; XX
OUT TR1
AND 613.03  ; Toerrkj. P4501
MOV(021) &600 D3198
LD TR1
ANDNOT 613.03  ; Toerrkj. P4501
MOV(021) &1000 D3198
LD TR0
AND P4501_UT
MOV(021) D3198 D7742  ; C_TYPE_VASK
LD TR0
ANDNOT P4501_UT
MOV(021) &0 D7742  ; C_TYPE_VASK
LD TR0
ANDNOT P_On
AND 589.00  ; PGM 589_DRIFT
OUT TR1
AND 613.03  ; Toerrkj. P4501
MOV(021) &600 D3198
LD TR1
ANDNOT 613.03  ; Toerrkj. P4501
MOV(021) &1000 D3198
LD TR0
ANDNOT P4501_UT
MOV(021) &0 D3198
; rung 19: FEIL PÅ SLANGESENSOR TRAKT UHT
LDNOT P_On
ANDNOT N5_B4201_SLANGKONTR  ; SLANGEKONTROLL VED TRAKT T27.42
OUT 615.15  ; Slangefeil Trakt UHT
; rung 20: Ingen_kommentar_funnet

### Section PAST21_TEMP_OG_NIVÅ

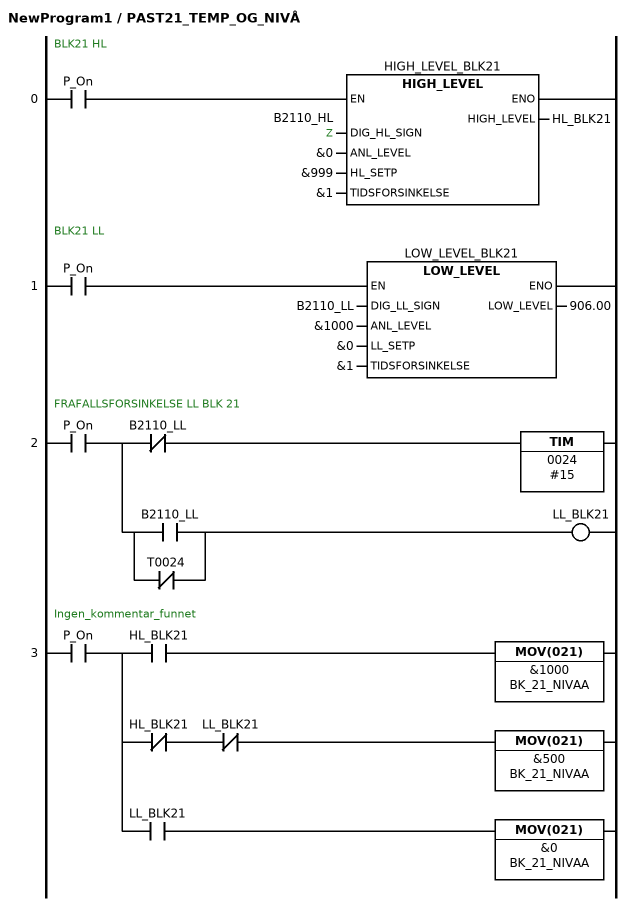
; rung 0: BLK21 HL
LD P_On
CALL HIGH_LEVEL_BLK21 : HIGH_LEVEL (DIG_HL_SIGN := B2110_HL, ANL_LEVEL := &0, HL_SETP := &999, TIDSFORSINKELSE := &1, HIGH_LEVEL => HL_BLK21)  ; Z
; rung 1: BLK21 LL
LD P_On
CALL LOW_LEVEL_BLK21 : LOW_LEVEL (DIG_LL_SIGN := B2110_LL, ANL_LEVEL := &1000, LL_SETP := &0, TIDSFORSINKELSE := &1, LOW_LEVEL => 906.00)
; rung 2: FRAFALLSFORSINKELSE LL BLK 21
LD P_On
OUT TR0
ANDNOT B2110_LL
TIM 0024 #15
LD TR0
LD B2110_LL
ORNOT T0024
ANDLD
OUT LL_BLK21
; rung 3: Ingen_kommentar_funnet
LD P_On
OUT TR0
AND HL_BLK21
MOV(021) &1000 BK_21_NIVAA
LD TR0
ANDNOT HL_BLK21
ANDNOT LL_BLK21
MOV(021) &500 BK_21_NIVAA
LD TR0
AND LL_BLK21
MOV(021) &0 BK_21_NIVAA
; rung 4: Ingen_kommentar_funnet

### Section PAST21_DRIFT_OG_TYPE_MELK

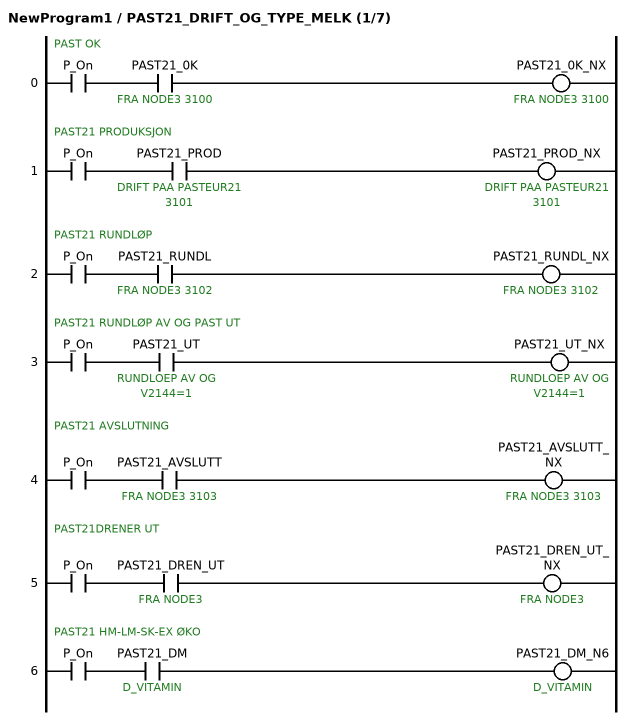
; rung 0: PAST OK
LD P_On
AND PAST21_0K  ; FRA NODE3 3100
OUT PAST21_0K_NX  ; FRA NODE3 3100
; rung 1: PAST21 PRODUKSJON
LD P_On
AND PAST21_PROD  ; DRIFT PAA PASTEUR21 3101
OUT PAST21_PROD_NX  ; DRIFT PAA PASTEUR21 3101
; rung 2: PAST21 RUNDLØP
LD P_On
AND PAST21_RUNDL  ; FRA NODE3 3102
OUT PAST21_RUNDL_NX  ; FRA NODE3 3102
; rung 3: PAST21 RUNDLØP AV OG PAST UT
LD P_On
AND PAST21_UT  ; RUNDLOEP AV OG V2144=1
OUT PAST21_UT_NX  ; RUNDLOEP AV OG V2144=1
; rung 4: PAST21 AVSLUTNING
LD P_On
AND PAST21_AVSLUTT  ; FRA NODE3 3103
OUT PAST21_AVSLUTT_NX  ; FRA NODE3 3103
; rung 5: PAST21DRENER UT
LD P_On
AND PAST21_DREN_UT  ; FRA NODE3
OUT PAST21_DREN_UT_NX  ; FRA NODE3
; rung 6: PAST21 HM-LM-SK-EX ØKO
LD P_On
AND PAST21_DM  ; D_VITAMIN
OUT PAST21_DM_N6  ; D_VITAMIN

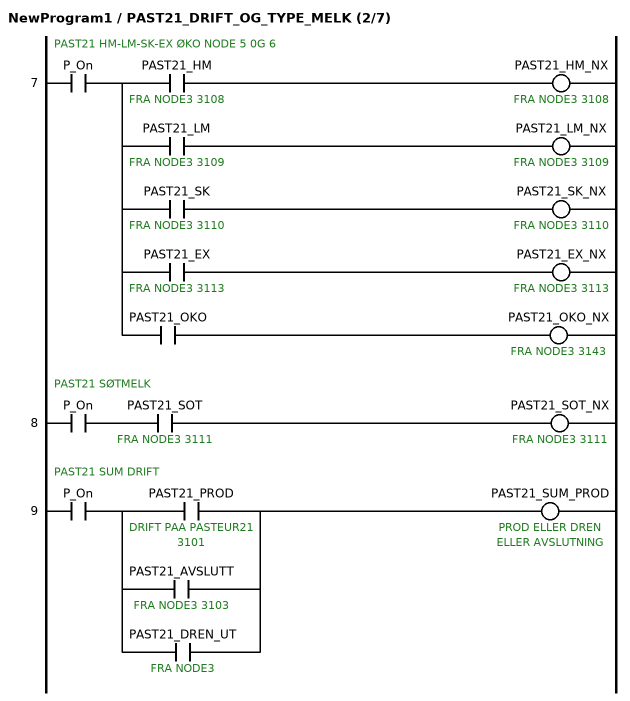
; rung 7: PAST21 HM-LM-SK-EX ØKO NODE 5 0G 6
LD P_On
OUT TR0
AND PAST21_HM  ; FRA NODE3 3108
OUT PAST21_HM_NX  ; FRA NODE3 3108
LD TR0
AND PAST21_LM  ; FRA NODE3 3109
OUT PAST21_LM_NX  ; FRA NODE3 3109
LD TR0
AND PAST21_SK  ; FRA NODE3 3110
OUT PAST21_SK_NX  ; FRA NODE3 3110
LD TR0
AND PAST21_EX  ; FRA NODE3 3113
OUT PAST21_EX_NX  ; FRA NODE3 3113
LD TR0
AND PAST21_OKO
OUT PAST21_OKO_NX  ; FRA NODE3 3143
; rung 8: PAST21 SØTMELK
LD P_On
AND PAST21_SOT  ; FRA NODE3 3111
OUT PAST21_SOT_NX  ; FRA NODE3 3111
; rung 9: PAST21 SUM DRIFT
LD P_On
LD PAST21_PROD  ; DRIFT PAA PASTEUR21 3101
OR PAST21_AVSLUTT  ; FRA NODE3 3103
OR PAST21_DREN_UT  ; FRA NODE3
ANDLD
OUT PAST21_SUM_PROD  ; PROD ELLER DREN ELLER AVSLUTNING

